FUNCTION_BLOCK EL3201
VAR
	_io : EL3xx1_Data;
	{attribute addProperty Name "WcState"}
	_wcState : WcStateInputToggle;
	{attribute addProperty Name "Info data"}
	_infoData : InfoDataAds;
END_VAR

PROPERTY IO : REFERENCE TO EL3xx1_Data
GET
IO REF= _io;
END_GET
END_PROPERTY

PROPERTY WcState : REFERENCE TO WcStateInputToggle
GET
WcState REF= _wcState;
END_GET
END_PROPERTY

END_FUNCTION_BLOCK

(* stored: Version 1.1.0.1, ProductVersion 3.1.4024.9
   POU EL3201: Id {99f09192-2418-0ba6-336f-1aab53325abf}, SpecialFunc None
   Property IO: Id {dbe293d1-e2d9-0d09-0725-f29fa7c4d563}
   Get Get: Id {c0be6323-1465-000b-1757-7ef1f7386845}
   Property WcState: Id {22c14b4a-41f3-05f9-1dfb-750234383bc8}
   Get Get: Id {17381bad-d822-0d75-2fed-ad94d2bb1541} *)
